// TwinCAT 3 PLC project XmlDOMPLC
// ProgramVersion: 3.1.4024.0
// libraries:
//   Tc2_Standard, * (Beckhoff Automation GmbH)
//   Tc2_System, * (Beckhoff Automation GmbH)
//   Tc2_Utilities, * (Beckhoff Automation GmbH)
//   Tc3_JsonXml, * (Beckhoff Automation GmbH)
//   Tc3_Module, * (Beckhoff Automation GmbH)
// project tree:
//   DUTs/ ST_Device.TcDUT
//   GVLs/ Globals.TcGVL (not stored)
//   / PlcTask.TcTTO (not stored)
//   POUs/ MAIN.TcPOU
// real-time tasks:
//   TASK PlcTask: cycle T#1ms, priority 20, ADS port 350

// ---- DUTs/ST_Device.TcDUT
TYPE ST_Device :
STRUCT
	value : DINT;
END_STRUCT
END_TYPE

// ---- POUs/MAIN.TcPOU
PROGRAM MAIN
VAR
	
  fbXml : FB_XmlDomParser;
  xmlDoc : SXmlNode;
  xmlConfig : SXmlNode;
  xmlParam : SXmlNode;
  xmlIterator : SXmlIterator;
  xmlParamNode : SXmlNode;
  xmlParamNodeValue : STRING;
  xmlParamNodeADSType : STRING;
  xmlParamNodePath : STRING;
		
	sMessageToParse : STRING(255) := '<Config><Parameter Path="device_1.value" ADSType="DINT">42</Parameter><Parameter Path="device_2.value" ADSType="DINT">24</Parameter></Config>';
	nState : INT := 0;
	
END_VAR



CASE nState OF 

	0 : (* Load XML content *)
			xmlDoc := fbXml.ParseDocument(sMessageToParse);
			nState := nState + 1;
			
	1:
			(* Parse XML nodes *)
			xmlConfig := fbXml.ChildByName(xmlDoc, 'Config');
			xmlIterator := fbXml.Begin(xmlConfig);
			nState := nState + 1;
					
	2:	IF (fbXml.IsEnd(xmlIterator)) THEN 
				nState:= nState +1; 
			ELSE
				xmlParamNode := fbXml.Node(xmlIterator);
  			xmlParamNodePath :=  fbXml.AttributeText(fbXml.Attribute(n:= xmlParamNode, name:='Path'));
  			xmlParamNodeADSType := fbXml.AttributeText(fbXml.Attribute(n:= xmlParamNode, name:='ADSType'));
  			xmlParamNodeValue := fbXml.NodeText(xmlParamNode);	
  			xmlIterator := fbXml.Next(xmlIterator);							
			END_IF
 		
	3:
			xmlIterator := fbXml.End(xmlConfig);
			nState := nState + 1;
			
	4:
			// Error, Done
	
END_CASE

END_PROGRAM
